// TIA Portal V17 export
// export: Created 2025-03-05T07:59:16.2029456Z, ExportSetting WithDefaults, DisplayName Totally Integrated Automation Portal, DisplayVersion V17 Update 8, DisplayName TIA Portal Openness, DisplayVersion V17 Update 8, DisplayName TIA Portal Version Control Interface, DisplayVersion V17, DisplayName SINAMICS Startdrive Advanced, DisplayVersion V17 SP2, DisplayName SINAMICS Startdrive G110M, G120, G120C, G120D, G120P, G115D, DisplayVersion V17 SP2, DisplayName SINAMICS Startdrive G130, G150, S120, S150, SINAMICS MV, S210, DisplayVersion V17 SP2, DisplayName STEP 7 Professional, DisplayVersion V17 Update 8, DisplayName SINUMERIK ONE STEP 7 Toolbox, DisplayVersion V17 Update 12, DisplayName SINUMERIK 840D sl STEP 7 Toolbox, DisplayVersion V17 Update 12, DisplayName STEP 7 Safety, DisplayVersion V17 Update 6, DisplayName WinCC Advanced, DisplayVersion V17 Update 8
FUNCTION "FC7000_SAFETY_DOORS" : Void   // FC7000, LAD
{ S7_Optimized_Access := 'FALSE' }
AUTHOR : ETXETAR
VERSION : 1.0
// stored: AutoNumber false, IsIECCheckEnabled false, SetENOAutomatically false, UDAEnableTagReadback false
BEGIN

REGION Network 1: CALL FC7002 UNIT 01 STATION 2 SAFETY DOOR
   // 2#0000_0001 OPTIONS 0 BIT 0 IMMEDIATE STOP REACTION OPTION
   // 2#0000_0010 OPTIONS 0 BIT 1 SEOC WARNING REACTION OPTION
   // 2#0000_0100 OPTIONS 0 BIT 2 CLOSED SENSOR INPUT OPTION
   // 2#0000_1000 OPTIONS 0 BIT 3 CIRCUIT E2 OPTION
   // 2#0001_0000 OPTIONS 0 BIT 4 HYDRAULIC DRIVE OPTION
   // 2#0010_0000 OPTIONS 0 BIT 5 CHIP CONVEYOR OPTION
   // 2#0100_0000 OPTIONS 0 BIT 6 SPARE OPTION
   // 2#1000_0000 OPTIONS 0 BIT 7 SPARE OPTION
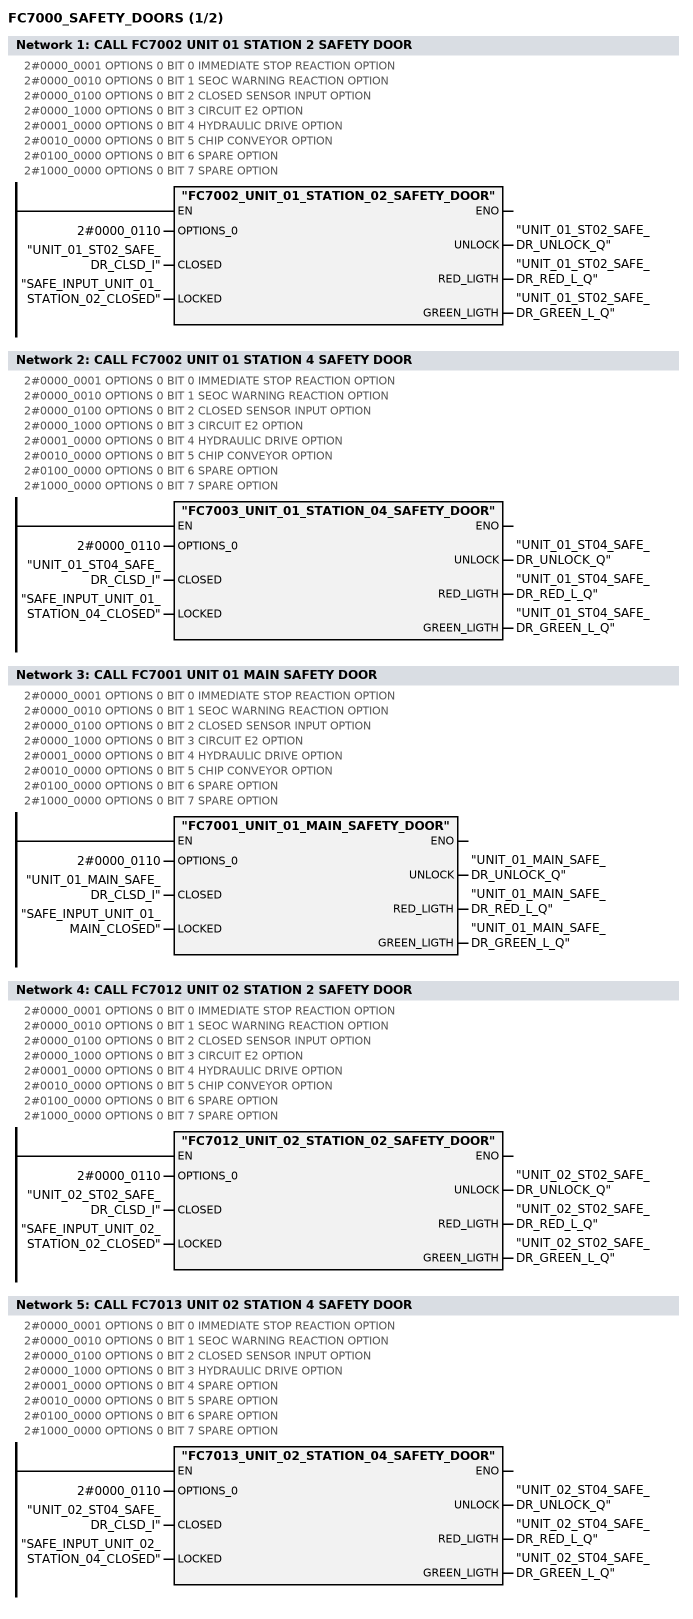
   RUNG wire#powerrail
      "FC7002_UNIT_01_STATION_02_SAFETY_DOOR"(OPTIONS_0 := 2#0000_0110, CLOSED := "UNIT_01_ST02_SAFE_DR_CLSD_I", LOCKED := "SAFE_INPUT_UNIT_01_STATION_02_CLOSED", UNLOCK => "UNIT_01_ST02_SAFE_DR_UNLOCK_Q", RED_LIGTH => "UNIT_01_ST02_SAFE_DR_RED_L_Q", GREEN_LIGTH => "UNIT_01_ST02_SAFE_DR_GREEN_L_Q")
   END_RUNG
   // the same network as SCL:
   "FC7002_UNIT_01_STATION_02_SAFETY_DOOR"(OPTIONS_0 := 2#0000_0110,
                           CLOSED := "UNIT_01_ST02_SAFE_DR_CLSD_I",
                           LOCKED := "SAFE_INPUT_UNIT_01_STATION_02_CLOSED",
                           UNLOCK => "UNIT_01_ST02_SAFE_DR_UNLOCK_Q",
                           RED_LIGTH => "UNIT_01_ST02_SAFE_DR_RED_L_Q",
                           GREEN_LIGTH => "UNIT_01_ST02_SAFE_DR_GREEN_L_Q");
END_REGION

REGION Network 2: CALL FC7002 UNIT 01 STATION 4 SAFETY DOOR
   // 2#0000_0001 OPTIONS 0 BIT 0 IMMEDIATE STOP REACTION OPTION
   // 2#0000_0010 OPTIONS 0 BIT 1 SEOC WARNING REACTION OPTION
   // 2#0000_0100 OPTIONS 0 BIT 2 CLOSED SENSOR INPUT OPTION
   // 2#0000_1000 OPTIONS 0 BIT 3 CIRCUIT E2 OPTION
   // 2#0001_0000 OPTIONS 0 BIT 4 HYDRAULIC DRIVE OPTION
   // 2#0010_0000 OPTIONS 0 BIT 5 CHIP CONVEYOR OPTION
   // 2#0100_0000 OPTIONS 0 BIT 6 SPARE OPTION
   // 2#1000_0000 OPTIONS 0 BIT 7 SPARE OPTION
   RUNG wire#powerrail
      "FC7003_UNIT_01_STATION_04_SAFETY_DOOR"(OPTIONS_0 := 2#0000_0110, CLOSED := "UNIT_01_ST04_SAFE_DR_CLSD_I", LOCKED := "SAFE_INPUT_UNIT_01_STATION_04_CLOSED", UNLOCK => "UNIT_01_ST04_SAFE_DR_UNLOCK_Q", RED_LIGTH => "UNIT_01_ST04_SAFE_DR_RED_L_Q", GREEN_LIGTH => "UNIT_01_ST04_SAFE_DR_GREEN_L_Q")
   END_RUNG
   // the same network as SCL:
   "FC7003_UNIT_01_STATION_04_SAFETY_DOOR"(OPTIONS_0 := 2#0000_0110,
                           CLOSED := "UNIT_01_ST04_SAFE_DR_CLSD_I",
                           LOCKED := "SAFE_INPUT_UNIT_01_STATION_04_CLOSED",
                           UNLOCK => "UNIT_01_ST04_SAFE_DR_UNLOCK_Q",
                           RED_LIGTH => "UNIT_01_ST04_SAFE_DR_RED_L_Q",
                           GREEN_LIGTH => "UNIT_01_ST04_SAFE_DR_GREEN_L_Q");
END_REGION

REGION Network 3: CALL FC7001 UNIT 01 MAIN SAFETY DOOR
   // 2#0000_0001 OPTIONS 0 BIT 0 IMMEDIATE STOP REACTION OPTION
   // 2#0000_0010 OPTIONS 0 BIT 1 SEOC WARNING REACTION OPTION
   // 2#0000_0100 OPTIONS 0 BIT 2 CLOSED SENSOR INPUT OPTION
   // 2#0000_1000 OPTIONS 0 BIT 3 CIRCUIT E2 OPTION
   // 2#0001_0000 OPTIONS 0 BIT 4 HYDRAULIC DRIVE OPTION
   // 2#0010_0000 OPTIONS 0 BIT 5 CHIP CONVEYOR OPTION
   // 2#0100_0000 OPTIONS 0 BIT 6 SPARE OPTION
   // 2#1000_0000 OPTIONS 0 BIT 7 SPARE OPTION
   RUNG wire#powerrail
      "FC7001_UNIT_01_MAIN_SAFETY_DOOR"(OPTIONS_0 := 2#0000_0110, CLOSED := "UNIT_01_MAIN_SAFE_DR_CLSD_I", LOCKED := "SAFE_INPUT_UNIT_01_MAIN_CLOSED", UNLOCK => "UNIT_01_MAIN_SAFE_DR_UNLOCK_Q", RED_LIGTH => "UNIT_01_MAIN_SAFE_DR_RED_L_Q", GREEN_LIGTH => "UNIT_01_MAIN_SAFE_DR_GREEN_L_Q")
   END_RUNG
   // the same network as SCL:
   "FC7001_UNIT_01_MAIN_SAFETY_DOOR"(OPTIONS_0 := 2#0000_0110,
                           CLOSED := "UNIT_01_MAIN_SAFE_DR_CLSD_I",
                           LOCKED := "SAFE_INPUT_UNIT_01_MAIN_CLOSED",
                           UNLOCK => "UNIT_01_MAIN_SAFE_DR_UNLOCK_Q",
                           RED_LIGTH => "UNIT_01_MAIN_SAFE_DR_RED_L_Q",
                           GREEN_LIGTH => "UNIT_01_MAIN_SAFE_DR_GREEN_L_Q");
END_REGION

REGION Network 4: CALL FC7012 UNIT 02 STATION 2 SAFETY DOOR
   // 2#0000_0001 OPTIONS 0 BIT 0 IMMEDIATE STOP REACTION OPTION
   // 2#0000_0010 OPTIONS 0 BIT 1 SEOC WARNING REACTION OPTION
   // 2#0000_0100 OPTIONS 0 BIT 2 CLOSED SENSOR INPUT OPTION
   // 2#0000_1000 OPTIONS 0 BIT 3 CIRCUIT E2 OPTION
   // 2#0001_0000 OPTIONS 0 BIT 4 HYDRAULIC DRIVE OPTION
   // 2#0010_0000 OPTIONS 0 BIT 5 CHIP CONVEYOR OPTION
   // 2#0100_0000 OPTIONS 0 BIT 6 SPARE OPTION
   // 2#1000_0000 OPTIONS 0 BIT 7 SPARE OPTION
   RUNG wire#powerrail
      "FC7012_UNIT_02_STATION_02_SAFETY_DOOR"(OPTIONS_0 := 2#0000_0110, CLOSED := "UNIT_02_ST02_SAFE_DR_CLSD_I", LOCKED := "SAFE_INPUT_UNIT_02_STATION_02_CLOSED", UNLOCK => "UNIT_02_ST02_SAFE_DR_UNLOCK_Q", RED_LIGTH => "UNIT_02_ST02_SAFE_DR_RED_L_Q", GREEN_LIGTH => "UNIT_02_ST02_SAFE_DR_GREEN_L_Q")
   END_RUNG
   // the same network as SCL:
   "FC7012_UNIT_02_STATION_02_SAFETY_DOOR"(OPTIONS_0 := 2#0000_0110,
                           CLOSED := "UNIT_02_ST02_SAFE_DR_CLSD_I",
                           LOCKED := "SAFE_INPUT_UNIT_02_STATION_02_CLOSED",
                           UNLOCK => "UNIT_02_ST02_SAFE_DR_UNLOCK_Q",
                           RED_LIGTH => "UNIT_02_ST02_SAFE_DR_RED_L_Q",
                           GREEN_LIGTH => "UNIT_02_ST02_SAFE_DR_GREEN_L_Q");
END_REGION

REGION Network 5: CALL FC7013 UNIT 02 STATION 4 SAFETY DOOR
   // 2#0000_0001 OPTIONS 0 BIT 0 IMMEDIATE STOP REACTION OPTION
   // 2#0000_0010 OPTIONS 0 BIT 1 SEOC WARNING REACTION OPTION
   // 2#0000_0100 OPTIONS 0 BIT 2 CLOSED SENSOR INPUT OPTION
   // 2#0000_1000 OPTIONS 0 BIT 3 HYDRAULIC DRIVE OPTION
   // 2#0001_0000 OPTIONS 0 BIT 4 SPARE OPTION
   // 2#0010_0000 OPTIONS 0 BIT 5 SPARE OPTION
   // 2#0100_0000 OPTIONS 0 BIT 6 SPARE OPTION
   // 2#1000_0000 OPTIONS 0 BIT 7 SPARE OPTION
   RUNG wire#powerrail
      "FC7013_UNIT_02_STATION_04_SAFETY_DOOR"(OPTIONS_0 := 2#0000_0110, CLOSED := "UNIT_02_ST04_SAFE_DR_CLSD_I", LOCKED := "SAFE_INPUT_UNIT_02_STATION_04_CLOSED", UNLOCK => "UNIT_02_ST04_SAFE_DR_UNLOCK_Q", RED_LIGTH => "UNIT_02_ST04_SAFE_DR_RED_L_Q", GREEN_LIGTH => "UNIT_02_ST04_SAFE_DR_GREEN_L_Q")
   END_RUNG
   // the same network as SCL:
   "FC7013_UNIT_02_STATION_04_SAFETY_DOOR"(OPTIONS_0 := 2#0000_0110,
                           CLOSED := "UNIT_02_ST04_SAFE_DR_CLSD_I",
                           LOCKED := "SAFE_INPUT_UNIT_02_STATION_04_CLOSED",
                           UNLOCK => "UNIT_02_ST04_SAFE_DR_UNLOCK_Q",
                           RED_LIGTH => "UNIT_02_ST04_SAFE_DR_RED_L_Q",
                           GREEN_LIGTH => "UNIT_02_ST04_SAFE_DR_GREEN_L_Q");
END_REGION

REGION Network 6: CALL FC7011 UNIT 02 MAIN SAFETY DOOR
   // 2#0000_0001 OPTIONS 0 BIT 0 IMMEDIATE STOP REACTION OPTION
   // 2#0000_0010 OPTIONS 0 BIT 1 SEOC WARNING REACTION OPTION
   // 2#0000_0100 OPTIONS 0 BIT 2 CLOSED SENSOR INPUT OPTION
   // 2#0000_1000 OPTIONS 0 BIT 3 CIRCUIT E2 OPTION
   // 2#0001_0000 OPTIONS 0 BIT 4 HYDRAULIC DRIVE OPTION
   // 2#0010_0000 OPTIONS 0 BIT 5 CHIP CONVEYOR OPTION
   // 2#0100_0000 OPTIONS 0 BIT 6 SPARE OPTION
   // 2#1000_0000 OPTIONS 0 BIT 7 SPARE OPTION
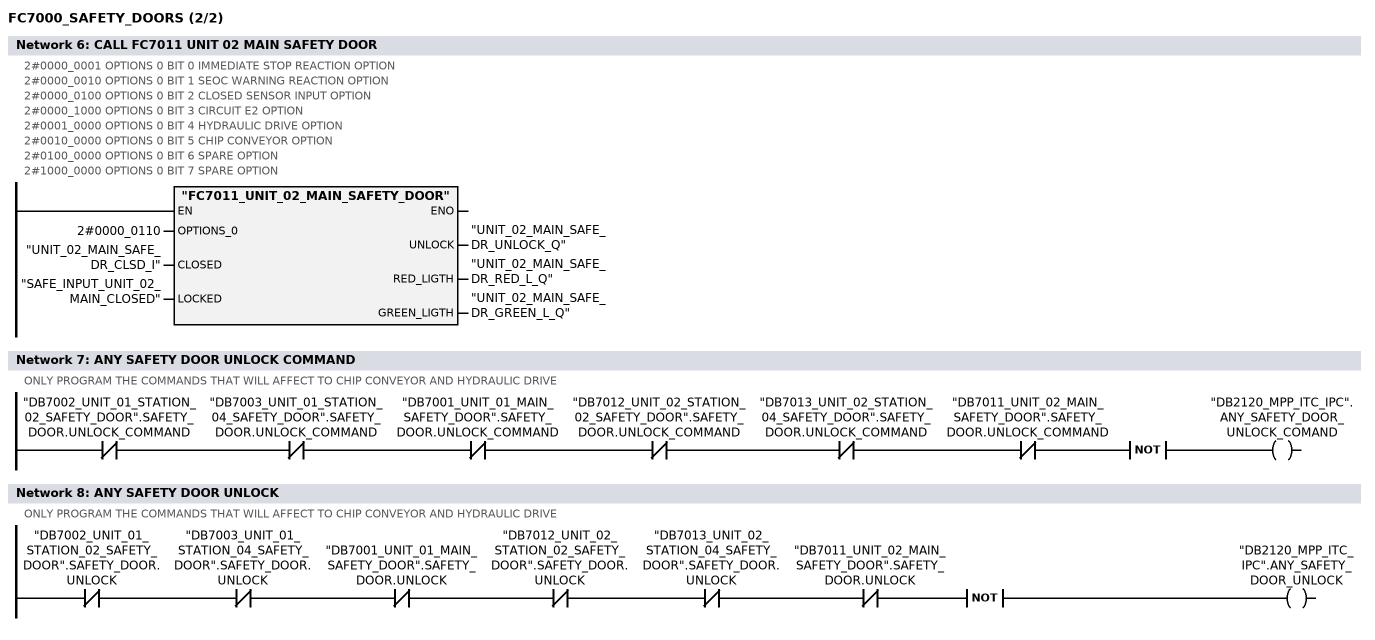
   RUNG wire#powerrail
      "FC7011_UNIT_02_MAIN_SAFETY_DOOR"(OPTIONS_0 := 2#0000_0110, CLOSED := "UNIT_02_MAIN_SAFE_DR_CLSD_I", LOCKED := "SAFE_INPUT_UNIT_02_MAIN_CLOSED", UNLOCK => "UNIT_02_MAIN_SAFE_DR_UNLOCK_Q", RED_LIGTH => "UNIT_02_MAIN_SAFE_DR_RED_L_Q", GREEN_LIGTH => "UNIT_02_MAIN_SAFE_DR_GREEN_L_Q")
   END_RUNG
   // the same network as SCL:
   "FC7011_UNIT_02_MAIN_SAFETY_DOOR"(OPTIONS_0 := 2#0000_0110,
                           CLOSED := "UNIT_02_MAIN_SAFE_DR_CLSD_I",
                           LOCKED := "SAFE_INPUT_UNIT_02_MAIN_CLOSED",
                           UNLOCK => "UNIT_02_MAIN_SAFE_DR_UNLOCK_Q",
                           RED_LIGTH => "UNIT_02_MAIN_SAFE_DR_RED_L_Q",
                           GREEN_LIGTH => "UNIT_02_MAIN_SAFE_DR_GREEN_L_Q");
END_REGION

REGION Network 7: ANY SAFETY DOOR UNLOCK COMMAND
   // ONLY PROGRAM THE COMMANDS THAT WILL AFFECT TO CHIP CONVEYOR AND HYDRAULIC DRIVE
   RUNG wire#powerrail
      I_Contact( "DB7002_UNIT_01_STATION_02_SAFETY_DOOR".SAFETY_DOOR.UNLOCK_COMMAND )
      I_Contact( "DB7003_UNIT_01_STATION_04_SAFETY_DOOR".SAFETY_DOOR.UNLOCK_COMMAND )
      I_Contact( "DB7001_UNIT_01_MAIN_SAFETY_DOOR".SAFETY_DOOR.UNLOCK_COMMAND )
      I_Contact( "DB7012_UNIT_02_STATION_02_SAFETY_DOOR".SAFETY_DOOR.UNLOCK_COMMAND )
      I_Contact( "DB7013_UNIT_02_STATION_04_SAFETY_DOOR".SAFETY_DOOR.UNLOCK_COMMAND )
      I_Contact( "DB7011_UNIT_02_MAIN_SAFETY_DOOR".SAFETY_DOOR.UNLOCK_COMMAND )
      Not()
      Coil( "DB2120_MPP_ITC_IPC".ANY_SAFETY_DOOR_UNLOCK_COMAND )
   END_RUNG
   // the same network as SCL:
   "DB2120_MPP_ITC_IPC".ANY_SAFETY_DOOR_UNLOCK_COMAND := NOT (NOT "DB7002_UNIT_01_STATION_02_SAFETY_DOOR".SAFETY_DOOR.UNLOCK_COMMAND AND NOT "DB7003_UNIT_01_STATION_04_SAFETY_DOOR".SAFETY_DOOR.UNLOCK_COMMAND AND NOT "DB7001_UNIT_01_MAIN_SAFETY_DOOR".SAFETY_DOOR.UNLOCK_COMMAND AND NOT "DB7012_UNIT_02_STATION_02_SAFETY_DOOR".SAFETY_DOOR.UNLOCK_COMMAND AND NOT "DB7013_UNIT_02_STATION_04_SAFETY_DOOR".SAFETY_DOOR.UNLOCK_COMMAND AND NOT "DB7011_UNIT_02_MAIN_SAFETY_DOOR".SAFETY_DOOR.UNLOCK_COMMAND);
END_REGION

REGION Network 8: ANY SAFETY DOOR UNLOCK
   // ONLY PROGRAM THE COMMANDS THAT WILL AFFECT TO CHIP CONVEYOR AND HYDRAULIC DRIVE
   RUNG wire#powerrail
      I_Contact( "DB7002_UNIT_01_STATION_02_SAFETY_DOOR".SAFETY_DOOR.UNLOCK )
      I_Contact( "DB7003_UNIT_01_STATION_04_SAFETY_DOOR".SAFETY_DOOR.UNLOCK )
      I_Contact( "DB7001_UNIT_01_MAIN_SAFETY_DOOR".SAFETY_DOOR.UNLOCK )
      I_Contact( "DB7012_UNIT_02_STATION_02_SAFETY_DOOR".SAFETY_DOOR.UNLOCK )
      I_Contact( "DB7013_UNIT_02_STATION_04_SAFETY_DOOR".SAFETY_DOOR.UNLOCK )
      I_Contact( "DB7011_UNIT_02_MAIN_SAFETY_DOOR".SAFETY_DOOR.UNLOCK )
      Not()
      Coil( "DB2120_MPP_ITC_IPC".ANY_SAFETY_DOOR_UNLOCK )
   END_RUNG
   // the same network as SCL:
   "DB2120_MPP_ITC_IPC".ANY_SAFETY_DOOR_UNLOCK := NOT (NOT "DB7002_UNIT_01_STATION_02_SAFETY_DOOR".SAFETY_DOOR.UNLOCK AND NOT "DB7003_UNIT_01_STATION_04_SAFETY_DOOR".SAFETY_DOOR.UNLOCK AND NOT "DB7001_UNIT_01_MAIN_SAFETY_DOOR".SAFETY_DOOR.UNLOCK AND NOT "DB7012_UNIT_02_STATION_02_SAFETY_DOOR".SAFETY_DOOR.UNLOCK AND NOT "DB7013_UNIT_02_STATION_04_SAFETY_DOOR".SAFETY_DOOR.UNLOCK AND NOT "DB7011_UNIT_02_MAIN_SAFETY_DOOR".SAFETY_DOOR.UNLOCK);
END_REGION
END_FUNCTION
